{attribute 'qualified_only'}
VAR_GLOBAL
		EtherCAT_Master_EMxxxx : EtherCAT_Master_EMxxxx_E69B3047;
END_VAR

(* stored: Version 1.2.0.0, ProductVersion 3.1.4024.11
   GVL GVL_iXlinker: Id {b8b08180-188e-4e13-8513-e27e5679470a} *)
